// TwinCAT 3 PLC project Main
// ProgramVersion: 3.1.4023.0
// libraries:
//   Tc2_Standard, * (Beckhoff Automation GmbH)
//   Tc2_System, * (Beckhoff Automation GmbH)
//   Tc3_Module, * (Beckhoff Automation GmbH)
// project tree:
//   / PlcTask.TcTTO
//   POUs/ I_Module.TcIO, I_Sensor.TcIO, I_VisitModules.TcIO, I_VisitSensors.TcIO, MAIN.TcPOU, Module.TcPOU, Sensor.TcPOU, StatusToStringLogVisitor.TcPOU, StatusToStringLogPrinterVisitor.TcPOU
// real-time tasks:
//   TASK PlcTask: cycle T#10ms, priority 20, ADS port 350

CONFIGURATION Main
    RESOURCE PLC ON TwinCAT3
        TASK PlcTask(INTERVAL := T#10ms, PRIORITY := 20);
        PROGRAM MAIN WITH PlcTask : MAIN;
    END_RESOURCE
END_CONFIGURATION

// ---- POUs/I_Module.TcIO
INTERFACE I_Module

METHOD PUBLIC GetLastErrorMessage : T_MAXSTRING
VAR_INPUT
END_VAR
END_METHOD

PROPERTY PUBLIC HasError : BOOL
GET
END_GET
END_PROPERTY

PROPERTY PUBLIC Name : T_MAXSTRING
GET
END_GET
END_PROPERTY

END_INTERFACE

// ---- POUs/I_Sensor.TcIO
INTERFACE I_Sensor

PROPERTY PUBLIC Name : T_MAXSTRING
GET
END_GET
END_PROPERTY

END_INTERFACE

// ---- POUs/I_VisitModules.TcIO
INTERFACE I_VisitModules

METHOD VisitModule
VAR_INPUT
	Module : I_Module;
END_VAR
END_METHOD

END_INTERFACE

// ---- POUs/I_VisitSensors.TcIO
INTERFACE I_VisitSensors

METHOD VisitSensor
VAR_INPUT
	Sensor : I_Sensor;
END_VAR
END_METHOD

END_INTERFACE

// ---- POUs/MAIN.TcPOU
PROGRAM MAIN
VAR
	initalised : BOOL := FALSE;
	
	infeedModule : Module(Name := 'infeed');
	processModule : Module(Name := 'process');
	outfeedModule : Module(Name := 'outfeed');
	
	jamSensor : Sensor(Name := 'outfeedJam');
	
	statusToStringLogVisitor : StatusToStringLogVisitor(status);
	statusToStringLogPrinterVisitor : StatusToStringLogPrinterVisitor(statusForPrinter);
	
	status : T_MAXSTRING;	
	statusForPrinter : T_MAXSTRING;	

END_VAR

IF NOT initalised THEN
	
	initalised := TRUE;
	infeedModule.SetError('Infeed Jammed');

END_IF

status := '';
statusForPrinter := '';

infeedModule.Accept(statusToStringLogVisitor);
processModule.Accept(statusToStringLogVisitor);

infeedModule.Accept(statusToStringLogPrinterVisitor);
processModule.Accept(statusToStringLogPrinterVisitor);
outfeedModule.Accept(statusToStringLogPrinterVisitor);

jamSensor.Accept(statusToStringLogPrinterVisitor);

END_PROGRAM

// ---- POUs/Module.TcPOU
FUNCTION_BLOCK Module IMPLEMENTS I_Module
VAR
	_name : T_MAXSTRING;
	_hasError : BOOL;
	lastErrorMessage : T_MAXSTRING;
END_VAR

METHOD PUBLIC Accept
VAR_INPUT
	Visitor : I_VisitModules;
END_VAR
Visitor.VisitModule(this^);
END_METHOD

METHOD FB_init : BOOL
VAR_INPUT
	bInitRetains : BOOL; // if TRUE, the retain variables are initialized (warm start / cold start)
	bInCopyCode : BOOL;  // if TRUE, the instance afterwards gets moved into the copy code (online change)
	Name : T_MAXSTRING;
END_VAR
_name := Name;
END_METHOD

METHOD PUBLIC GetLastErrorMessage : T_MAXSTRING
VAR_INPUT
END_VAR
GetLastErrorMessage := lastErrorMessage;
END_METHOD

PROPERTY PUBLIC HasError : BOOL
GET
HasError := _hasError;
END_GET
END_PROPERTY

PROPERTY PUBLIC Name : T_MAXSTRING
GET
Name := _name;
END_GET
END_PROPERTY

METHOD PUBLIC SetError
VAR_INPUT
	Message : T_Maxstring;
END_VAR
lastErrorMessage := Message;
_hasError := TRUE;
END_METHOD

END_FUNCTION_BLOCK

// ---- POUs/Sensor.TcPOU
FUNCTION_BLOCK Sensor IMPLEMENTS I_Sensor
VAR
	_name : T_MAXSTRING;
END_VAR

METHOD PUBLIC Accept
VAR_INPUT
	Visitor : I_VisitSensors;
END_VAR
Visitor.VisitSensor(this^);
END_METHOD

METHOD FB_init : BOOL
VAR_INPUT
	bInitRetains : BOOL; // if TRUE, the retain variables are initialized (warm start / cold start)
	bInCopyCode : BOOL;  // if TRUE, the instance afterwards gets moved into the copy code (online change)
	Name : T_MAXSTRING;
END_VAR
_name := Name;
END_METHOD

PROPERTY PUBLIC Name : T_MAXSTRING
GET
Name := _name;
END_GET
END_PROPERTY

END_FUNCTION_BLOCK

// ---- POUs/StatusToStringLogVisitor.TcPOU
FUNCTION_BLOCK StatusToStringLogVisitor IMPLEMENTS I_VisitModules
VAR
	stringLog : REFERENCE TO T_MAXSTRING;
END_VAR

METHOD FB_init : BOOL
VAR_INPUT
	bInitRetains : BOOL; // if TRUE, the retain variables are initialized (warm start / cold start)
	bInCopyCode : BOOL;  // if TRUE, the instance afterwards gets moved into the copy code (online change)
	StringLog : REFERENCE TO T_MAXSTRING;
END_VAR
this^.stringLog REF= StringLog;
END_METHOD

METHOD VisitModule
VAR_INPUT
	Module : I_Module;
END_VAR
stringLog := concat(stringLog, '[');
stringLog := concat(stringLog, Module.Name);
stringLog := concat(stringLog, ']');

IF Module.HasError THEN
	stringLog := concat(stringLog, ': Has Error ');
	stringLog := concat(stringLog, Module.GetLastErrorMessage());
	stringLog := concat(stringLog, '. ');
ELSE
	stringLog := concat(stringLog, ': Has No Error. ');
END_IF
END_METHOD

END_FUNCTION_BLOCK

// ---- POUs/StatusToStringLogPrinterVisitor.TcPOU
FUNCTION_BLOCK StatusToStringLogPrinterVisitor IMPLEMENTS I_VisitModules, I_VisitSensors
VAR
	stringLog : REFERENCE TO T_MAXSTRING;
END_VAR

METHOD FB_init : BOOL
VAR_INPUT
	bInitRetains : BOOL; // if TRUE, the retain variables are initialized (warm start / cold start)
	bInCopyCode : BOOL;  // if TRUE, the instance afterwards gets moved into the copy code (online change)
	StringLog : REFERENCE TO T_MAXSTRING;
END_VAR
this^.stringLog REF= StringLog;
END_METHOD

METHOD VisitModule
VAR_INPUT
	Module : I_Module;
END_VAR
IF Module.HasError THEN
	RETURN;
END_IF

stringLog := concat(stringLog, '?');
stringLog := concat(stringLog, Module.Name);
stringLog := concat(stringLog, '?');
END_METHOD

METHOD VisitSensor
VAR_INPUT
	Sensor : I_Sensor;
END_VAR
stringLog := concat(stringLog, '<sensor name:=');
stringLog := concat(stringLog, Sensor.Name);
stringLog := concat(stringLog, '>');
END_METHOD

END_FUNCTION_BLOCK
